(* CoDeSys 2.3 export: PLC_PRG.EXP *)

(* POU PLC_PRG, ST *)
PROGRAM PLC_PRG
VAR
END_VAR
GEMMA();

(*Simulaciones*)
Carrito_Rojo;
Carrito_Verde;
Cambio_Escenas;
Luces;
Simulacion_Almacen;
END_PROGRAM
